FUNCTION_BLOCK EL4134
VAR
	_io : EL4xx4_Data;
	{attribute addProperty Name "WcState"}
	_wcState : WcStateBase;
	{attribute addProperty Name "Info data"}
	_infoData : InfoDataAds;
END_VAR

PROPERTY IO : REFERENCE TO EL4xx4_Data
GET
IO REF= _io;
END_GET
END_PROPERTY

PROPERTY WcState : REFERENCE TO WcStateBase
GET
WcState REF= _wcState;
END_GET
END_PROPERTY

END_FUNCTION_BLOCK

(* stored: Version 1.1.0.1, ProductVersion 3.1.4024.9
   POU EL4134: Id {6384e766-3180-056a-37be-31fe887a1008}, SpecialFunc None
   Property IO: Id {b272ec04-1466-0392-0593-499a591a2e88}
   Get Get: Id {c5698d0f-4ec8-03e4-2ba9-06d32170a959}
   Property WcState: Id {d4e051ea-f771-0782-010b-8cfb5800438d}
   Get Get: Id {b2c7d398-523e-0289-211e-43ca74928135} *)
